// TIA Portal project "s" (V18)

(* hardware
DEVICE "S7-1200 station_1"  S7-1200 Station
   slot 0: "Rack_0"  S7-1200 Rack  Rack  V1.0
   slot 1: "PLC_1"  CPU 1214C DC/DC/DC  6ES7 214-1AG40-0XB0  V4.6
*)

// ===== PLC "PLC_1"  CPU 1214C DC/DC/DC =====

VAR_GLOBAL   // PLC tag table "Default tag table"
   "Tag_1" AT %QB0 : Byte;
   "Tag_2" AT %I0.0 : Bool;
   "Tag_3" AT %Q0.1 : Bool;
   "Tag_4" AT %MW64 : Int;
   "System_Byte" AT %MB21 : Byte;
   "FirstScan" AT %M21.0 : Bool;
   "DiagStatusUpdate" AT %M21.1 : Bool;
   "AlwaysTRUE" AT %M21.2 : Bool;
   "AlwaysFALSE" AT %M21.3 : Bool;
END_VAR

ORGANIZATION_BLOCK "Main"   // OB1, LAD, ProgramCycle
TITLE = "Main Program Sweep (Cycle)"
{ S7_Optimized_Access := 'TRUE' }
VERSION : 0.1
   VAR_INPUT
      Initial_Call : Bool;   // Initial call of this OB
      Remanence : Bool;   // =True, if remanent data are available
   END_VAR
BEGIN
END_ORGANIZATION_BLOCK

ORGANIZATION_BLOCK "startup_OB"   // OB100, LAD, Startup
TITLE = "Complete Restart"
{ S7_Optimized_Access := 'TRUE' }
VERSION : 0.1
// StartupOB
// Stop konumundan run konumuna geçtiğinde bir defa çalışır
   VAR_INPUT
      LostRetentive : Bool;   // True if retentive data are lost
      LostRTC : Bool;   // True if date and time are lost
   END_VAR
BEGIN

REGION Network 1
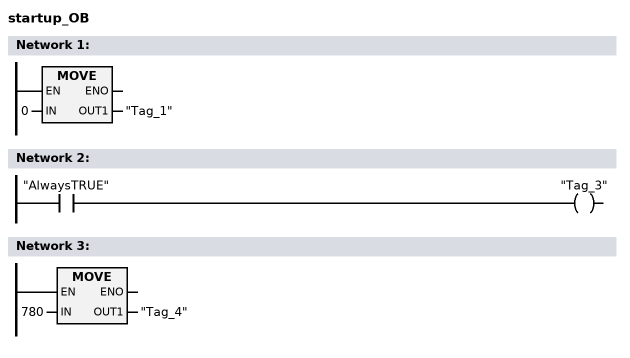
   RUNG wire#powerrail
      Move(in := 0, out1 => "Tag_1")
   END_RUNG
   // the same network as SCL:
   "Tag_1" := 0;
END_REGION

REGION Network 2
   RUNG wire#powerrail
      Contact( "AlwaysTRUE" )
      Coil( "Tag_3" )
   END_RUNG
   // the same network as SCL:
   "Tag_3" := "AlwaysTRUE";
END_REGION

REGION Network 3
   RUNG wire#powerrail
      Move(in := 780, out1 => "Tag_4")
   END_RUNG
   // the same network as SCL:
   "Tag_4" := 780;
END_REGION
END_ORGANIZATION_BLOCK